FUNCTION_BLOCK AUI_MUX_5 (* AUI multiplexor (generic FB) *)
  (* Standard: 61499-2; Description: Copyright (c) 2026 HR Agrartechnik GmbH This program and the accompanying materials are made available under the terms of the Eclipse Public License 2.0 which is available at https://www.eclipse.org/legal/epl-2.0/ SPDX-License-Identifier: EPL-2.0 *)
  (* Version 1.0, 2026-05-28, Franz Höpfinger, HR Agrartechnik GmbH *)
  PACKAGE adapter::selection::unidirectional;
  {SET_ATTRIBUTE(eclipse4diac::core::GenericClassName, 'GEN_AUI_MUX')}
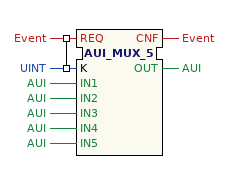
  EVENT_INPUT
    REQ WITH K; (* Set Index K *)
  END_EVENT
  EVENT_OUTPUT
    CNF; (* Confirmation of Set Index K *)
  END_EVENT
  VAR_INPUT
    K : UINT; (* index *)
  END_VAR
  SOCKETS
    IN1 : adapter::types::unidirectional::AUI; (* Input value 1 *)
    IN2 : adapter::types::unidirectional::AUI; (* Input value 2 *)
    IN3 : adapter::types::unidirectional::AUI; (* Input value 3 *)
    IN4 : adapter::types::unidirectional::AUI; (* Input value 4 *)
    IN5 : adapter::types::unidirectional::AUI; (* Input value 5 *)
  END_SOCKETS
  PLUGS
    OUT : adapter::types::unidirectional::AUI; (* IN1 for K = 0, IN2 for K = 1, IN3 for K = 2, IN4 for K = 3, IN5 for K = 4 *)
  END_PLUGS
END_FUNCTION_BLOCK
